# EPICS alarm handler configuration: mps_database/bareTest/alarms/areas/mpln_clts_mp01.alhConfig
GROUP NULL MPLN:CLTS:MP01:1
$ALIAS MPS Link Node 195
$GUIDANCE
LTUH MPS
   Group Name: MPLN:CLTS:MP01:1
   Summary PV:  MPLN:CLTS:MP01:1:STATSUMY
$END
CHANNEL  MPLN:CLTS:MP01:1    MPLN:CLTS:MP01:1:MPS_EN_RBV		-----
CHANNEL  MPLN:CLTS:MP01:1    MPLN:CLTS:MP01:1:LC1_MODE_RBV		-----
